GLOBALCONSTANTS IG4_NAME_Functions (* Industry Group 4 specific function defines *)
  (* Standard: 61499-1 *)
  (* Version 1.0, 2026-06-29, Franz Höpfinger, Demmler Andreas Fahrzeugbau *)
  PACKAGE isobus::pgn::const;
  VAR_GLOBAL CONSTANT
    F_ALARM_SYSTEM_CONTROL_FOR_MARINE_ENGINES : BYTE := 128; (* Sys: Non-specific System, Func: Alarm System Control for Marine Engines - The ECU that controls *)
    F_PROTECTION_SYSTEM_FOR_MARINE_ENGINES : BYTE := 129; (* Sys: Non-specific System, Func: Protection System for Marine Engines - The first ECU that *)
    F_DISPLAY_FOR_PROTECTION_SYSTEM_FOR_MARINE_ENGINES : BYTE := 130; (* Sys: Non-specific System, Func: Display for Protection System for Marine Engines - The ECU that *)
    F_NOT_AVAILABLE : BYTE := 255; (* Sys: Non-specific System, Func: Not Available - This assignment can be used until an explicit *)
    F_SYSTEM_TOOLS_NOT_AVAILABLE : BYTE := 255; (* Sys: System tools, Func: Not Available *)
    F_SAFETY_SYSTEMS_NOT_AVAILABLE : BYTE := 255; (* Sys: Safety systems, Func: Not Available *)
    F_GATEWAY : BYTE := 130; (* Sys: Gateway, Func: *)
    F_POWER_MGMT_LIGHTING_SWITCH : BYTE := 130; (* Sys: Power management and lighting systems, Func: Switch *)
    F_POWER_MGMT_LIGHTING_LOAD : BYTE := 140; (* Sys: Power management and lighting systems, Func: Load *)
    F_STEERING_SYSTEMS_FOLLOW_UP_CONTROLLER : BYTE := 130; (* Sys: Steering systems, Func: Follow-up Controller *)
    F_STEERING_SYSTEMS_MODE_CONTROLLER : BYTE := 140; (* Sys: Steering systems, Func: Mode Controller *)
    F_STEERING_SYSTEMS_AUTOMATIC_STEERING_CONTROLLER : BYTE := 150; (* Sys: Steering systems, Func: Automatic Steering Controller *)
    F_STEERING_SYSTEMS_HEADING_SENSORS : BYTE := 160; (* Sys: Steering systems, Func: Heading Sensors *)
    F_PROPULSION_SYSTEMS_ENGINEROOM_MONITORING : BYTE := 130; (* Sys: Propulsion systems, Func: Engineroom monitoring *)
    F_PROPULSION_SYSTEMS_ENGINE_INTERFACE : BYTE := 140; (* Sys: Propulsion systems, Func: Engine Interface *)
    F_PROPULSION_SYSTEMS_ENGINE_CONTROLLER : BYTE := 150; (* Sys: Propulsion systems, Func: Engine Controller *)
    F_PROPULSION_SYSTEMS_ENGINE_GATEWAY : BYTE := 160; (* Sys: Propulsion systems, Func: Engine Gateway *)
    F_PROPULSION_SYSTEMS_CONTROL_HEAD : BYTE := 170; (* Sys: Propulsion systems, Func: Control Head *)
    F_PROPULSION_SYSTEMS_ACTUATOR : BYTE := 180; (* Sys: Propulsion systems, Func: Actuator *)
    F_PROPULSION_SYSTEMS_GAUGE_INTERFACE : BYTE := 190; (* Sys: Propulsion systems, Func: Gauge Interface *)
    F_PROPULSION_SYSTEMS_GAUGE_LARGE : BYTE := 200; (* Sys: Propulsion systems, Func: Gauge Large *)
    F_PROPULSION_SYSTEMS_GAUGE_SMALL : BYTE := 210; (* Sys: Propulsion systems, Func: Gauge Small *)
    F_PROPULSION_SYSTEMS_PROPULSION_SENSORS_GATEWAY : BYTE := 220; (* Sys: Propulsion systems, Func: Propulsion Sensors & Gateway *)
    F_NAVIGATION_SYSTEMS_SOUNDER_DEPTH : BYTE := 130; (* Sys: Navigation systems, Func: Sounder, depth *)
    F_NAVIGATION_SYSTEMS : BYTE := 140; (* Sys: Navigation systems, Func: *)
    F_NAVIGATION_SYSTEMS_GLOBAL_NAVIGATION_SATELLITE_SYSTEM_GNSS : BYTE := 145; (* Sys: Navigation systems, Func: Global Navigation Satellite System (GNSS) *)
    F_NAVIGATION_SYSTEMS_LORAN_C : BYTE := 150; (* Sys: Navigation systems, Func: Loran C *)
    F_NAVIGATION_SYSTEMS_SPEED_SENSORS : BYTE := 155; (* Sys: Navigation systems, Func: Speed Sensors *)
    F_NAVIGATION_SYSTEMS_TURN_RATE_INDICATOR : BYTE := 160; (* Sys: Navigation systems, Func: Turn Rate Indicator *)
    F_NAVIGATION_SYSTEMS_INTEGRATED_NAVIGATION : BYTE := 170; (* Sys: Navigation systems, Func: Integrated Navigation *)
    F_NAVIGATION_SYSTEMS_RADAR_AND_OR_RADAR_PLOTTING : BYTE := 200; (* Sys: Navigation systems, Func: Radar and/or Radar Plotting *)
    F_NAVIGATION_SYSTEMS_ELECTRONIC_CHART_DISPLAY_INFORMATION_SYSTEM_ECDIS : BYTE := 205; (* Sys: Navigation systems, Func: Electronic Chart Display & Information System (ECDIS) *)
    F_NAVIGATION_SYSTEMS_ELECTRONIC_CHART_SYSTEM_ECS : BYTE := 210; (* Sys: Navigation systems, Func: Electronic Chart System (ECS) *)
    F_NAVIGATION_SYSTEMS_DIRECTION_FINDER : BYTE := 220; (* Sys: Navigation systems, Func: Direction Finder *)
    F_COMMUNICATIONS_SYSTEMS_EMERGENCY_POSITION_INDICATING_BEACON_EPIRB : BYTE := 130; (* Sys: Communications systems, Func: Emergency Position Indicating Beacon (EPIRB) *)
    F_COMMUNICATIONS_SYSTEMS_AUTOMATIC_IDENTIFICATION_SYSTEM : BYTE := 140; (* Sys: Communications systems, Func: Automatic Identification System *)
    F_COMMUNICATIONS_SYSTEMS_DIGITAL_SELECTIVE_CALLING_DSC : BYTE := 150; (* Sys: Communications systems, Func: Digital Selective Calling (DSC) *)
    F_COMMUNICATIONS_SYSTEMS_DATA_RECEIVER : BYTE := 160; (* Sys: Communications systems, Func: Data Receiver *)
    F_COMMUNICATIONS_SYSTEMS_SATELLITE : BYTE := 170; (* Sys: Communications systems, Func: Satellite *)
    F_COMMUNICATIONS_SYSTEMS_RADIO_TELEPHONE_MF_HF : BYTE := 180; (* Sys: Communications systems, Func: Radio-Telephone (MF/HF) *)
    F_COMMUNICATIONS_SYSTEMS_RADIO_TELEPHONE_VHF : BYTE := 190; (* Sys: Communications systems, Func: Radio-Telephone (VHF) *)
    F_INSTRUMENTATION_GENERAL_TIME_DATE_SYSTEMS : BYTE := 130; (* Sys: Instrumentation/general systems, Func: Time/Date systems *)
    F_INSTRUMENTATION_GENERAL_VOYAGE_DATA_RECORDER : BYTE := 140; (* Sys: Instrumentation/general systems, Func: Voyage Data Recorder *)
    F_INSTRUMENTATION_GENERAL_INTEGRATED_INSTRUMENTATION : BYTE := 150; (* Sys: Instrumentation/general systems, Func: Integrated Instrumentation *)
    F_INSTRUMENTATION_GENERAL_GENERAL_PURPOSE_DISPLAYS : BYTE := 160; (* Sys: Instrumentation/general systems, Func: General Purpose Displays *)
    F_INSTRUMENTATION_GENERAL_GENERAL_SENSOR_BOX : BYTE := 170; (* Sys: Instrumentation/general systems, Func: General Sensor Box *)
    F_INSTRUMENTATION_GENERAL_WEATHER_INSTRUMENTS : BYTE := 180; (* Sys: Instrumentation/general systems, Func: Weather Instruments *)
    F_INSTRUMENTATION_GENERAL_TRANSDUCER_GENERAL : BYTE := 190; (* Sys: Instrumentation/general systems, Func: Transducer/general *)
    F_INSTRUMENTATION_GENERAL_NMEA_0183_CONVERTER : BYTE := 200; (* Sys: Instrumentation/general systems, Func: NMEA 0183 Converter *)
    F_ENVIRONMENTAL_HVAC_NOT_AVAILABLE : BYTE := 255; (* Sys: Environmental (HVAC) systems, Func: Not Available *)
    F_DECK_CARGO_FISHING_NOT_AVAILABLE : BYTE := 255; (* Sys: Deck, cargo, and fishing equipment systems, Func: Not Available *)
  END_VAR
END_GLOBALCONSTANTS
